Staubli VAL3: PALLET.dtx

num nOldIndex
num nStep
string sInstruction
public string sItems
string sMessage
string sMenu
public bool bMoveType[3]
  [0] = true
  [1] = true
public bool bStepping
bool bToSave
string sTrajType
Trajectory tTraj
  [0]
    TrajectoryItem tSuper
      [0]
        num distance
        num moveType
        num nTime
        num nStop
        num nTcpAction
        string comment
        bool toStop
        mdesc nom_speed = {tmax=300, rmax=9999, leave=30, reach=30}
        InstrItem iInstr[3]
          [0]
            string sType
            string sData
          [1]
            string sType
            string sData
          [2]
            string sType
            string sData
        num nMoveId
    string sID
    num nId
mdesc mMdesc = {accel=10, vel=10, blend=off}
num nKey
frame fSetFrame = {fatherId=world[0]}
TrajPallet pEditPoint
  [0]
    TrajPointItem tData
      [0]
        TrajectoryItem tSuper
          [0]
            num distance
            num moveType
            num nTime
            num nStop
            num nTcpAction
            string comment
            bool toStop
            mdesc nom_speed = {tmax=600, rmax=9999, leave=30, reach=30}
            InstrItem iInstr[3]
              [0]
                string sType
                string sData
              [1]
                string sType
                string sData
              [2]
                string sType
                string sData
            num nMoveId
        pointRx pPoint = {fatherId=pEditPoint[0].fFrame[0]}
        num nType
    frame fFrame = {fatherId=pEditPoint[0].fReference[0]}
    num nIndexTool
    string sID
    trsf trAppro[2]
    trsf trDepart[2]
    num nX = 1
    num nY = 1
    num nZ = 1
    num nIndex
    num nDistanceXYZ[3]
      [0] = 1
      [1] = 1
      [2] = 1
    string sAction
    pointRx pO = {fatherId=pEditPoint[0].fReference[0]}
    pointRx pX = {fatherId=pEditPoint[0].fReference[0]}
    pointRx pY = {fatherId=pEditPoint[0].fReference[0]}
    pointRx pZ = {fatherId=pEditPoint[0].fReference[0]}
    num nSpeedApproach = 500
    num nSpeedDepart = 500
    num nIndexFrame
    frame fReference = {fatherId=world[0]}
string sTrajCycle
